TEXTLIST TXT_LIST_OBJECTS
  _3627.PLC_851.PrgStation.fbPowerAdapter1 = 'Netzteil 1' | de: 'Maschine' | en: 'Maschine'
  _3627.PLC_851.PrgStation.fbPowerAdapter2 = 'Netzteil 2' | de: 'Not-Halt links' | en: 'E-Stop left'
  _3627.PLC_851.PrgStation.fbZylinderLinks = 'Zylinder Links' | de: 'Not-Halt rechts' | en: 'E-Stop right'
  _3627.PLC_851.PrgStation.fbZylinderRechts = 'Zylinder Rechts' | de: 'Schutztür oben' | en: 'Door left'
  _3627.PLC_851.PrgStation.fbCalibrateVoltageInput1 = 'Scallieren Spannung (V)' | de: 'Schutztür rechts' | en: 'Door right'
  _3627.PLC_851.PrgStation.fbCalibrateVoltageInput2 = 'Scallieren Spannung (V)' | de: 'Maschine' | en: 'Machine'
  _3627.PLC_851.PrgStation.fbCalibrateCurrentInput1 = 'Scallieren Strom (A)' | de: 'Vakuum Druckstück' | en: 'Sensor 1'
  _3627.PLC_851.PrgStation.fbCalibrateCurrentInput2 = 'Scallieren Strom (A)' | de: 'Vakuum Druckpilz' | en: 'Vac Syst 1'
  _3531.PLC_851.PrgStation.fbStepSeqFindZeroPosPolepiece = 'Nullpunkt Suche Druckstück' | de: 'Nullpunkt-Suche Druckstück'
  _3531.PLC_851.PrgStation.fbStepSeqFindZeroPosPole = 'Nullpunkt Suche Stange' | de: 'Nullpunkt-Suche Stange'
  _3531.PLC_851.PrgStation.fbScanner = 'Scanner Druckstück' | de: 'Scanner Druckstück' | en: 'Scan Polepiece'
  _3531.PLC_851.PrgStation.fbECMaster = 'Beckoff PC' | de: 'Beckoff PC'
  _3531.PLC_851.PrgStation.fbPress = 'Kistler Presse' | de: 'Kistler Presse'
  _3531.PLC_851.PrgStation.fbCamera1 = 'Kamera Druckstange' | de: 'Kamera Druckstange' | en: 'Camera 1'
  _3531.PLC_851.PrgStation.fbCamera2 = 'Kamera Druckpilz' | de: 'Kamera Druckpilz' | en: 'Camera 2'
  _3531.PLC_851.PrgStation.fbGripper1 = 'Greifer links' | de: 'Greifer links'
  _3531.PLC_851.PrgStation.fbGripper2 = 'Greifer rechts' | de: 'Greifer rechts'
  _3531.PLC_851.PrgStation.fbAxisDruckstangeFunktions = 'Schrittmotor Druckstange' | de: 'Schrittmotor Druckstange'
  _3531.PLC_851.PrgStation.fbAxisDruckstueckFunctions = 'Schrittmotor Druckstück' | de: 'Schrittmotor Druckstück'
   = ''
END_TEXTLIST

(* stored: Version 1.1.0.1, ProductVersion 3.1.4024.9
   TextList TXT_LIST_OBJECTS: Id {dc98b7f5-a14b-47a3-9dde-dd7a9b8ee9ef} *)
